{attribute 'reflection'} 
FUNCTION_BLOCK FB_Teste
VAR
    {attribute 'instance-path'} 
    {attribute 'noinit'} 
	varTeste:STRING;
END_VAR

END_FUNCTION_BLOCK

(* stored: Version 1.1.0.1, ProductVersion 3.1.4024.12
   POU FB_Teste: Id {66e009f7-7c1e-46b8-ac1e-3cc645133fb7}, SpecialFunc None *)
